// TIA Portal project "FactoryIO_Template_S7-1200_V15_V15.1" (V15.1)
// Vorlageprojekt für das Buch mit Zielsystem S7-1200

(* hardware
DEVICE "S7-1200-Station_1"  S7-1200 Station
   slot 0: "Baugruppenträger_0"  Rack  V1.0
   slot 1: "PLC_1"  CPU 1211C DC/DC/DC  6ES7 211-1AE40-0XB0  V4.1
DEVICE "HMI_1"  KTP900 Basic PN
   slot 0: "HMI_1"  KTP900 Basic PN  6AV2 123-2JB03-0AX0  15.1.0.0
   slot 1: "HMI_RT_1"  KTP900 Basic PN  6AV2 123-2JB03-0AX0  15.1.0.0
   slot 5: "HMI_1.IE_CP_1"  PROFINET Interface  15.0.1.0
      slot 1: "PROFINET Interface_1"  PROFINET Interface
         slot 1: "Port_1"  Port
*)

// ===== PLC "PLC_1"  CPU 1211C DC/DC/DC =====

VAR_GLOBAL   // PLC tag table "Standard-Variablentabelle"
   "Moving X" AT %I0.0 : Bool;
   "Moving Z" AT %I0.1 : Bool;
   "Item detected" AT %I0.2 : Bool;
   "Lid at place" AT %I0.3 : Bool;
   "Lid clamped" AT %I0.4 : Bool;
   "Pos. at limit (lids)" AT %I0.5 : Bool;
   "Base at place" AT %I0.6 : Bool;
   "Base clamped" AT %I0.7 : Bool;
   "Pos. at limit (bases)" AT %I1.0 : Bool;
   "Part leaving" AT %I1.1 : Bool;
   "Start" AT %I1.2 : Bool;
   "Reset" AT %I1.3 : Bool;
   "Stop" AT %I1.4 : Bool;
   "Emergency stop" AT %I1.5 : Bool;
   "Auto" AT %I1.6 : Bool;
   "Running" AT %I1.7 : Bool;
   "Move X" AT %Q0.0 : Bool;
   "Move Z" AT %Q0.1 : Bool;
   "Grab" AT %Q0.2 : Bool;
   "Lids conveyor" AT %Q0.3 : Bool;
   "Clamp lid" AT %Q0.4 : Bool;
   "Pos. raise (lids)" AT %Q0.5 : Bool;
   "Bases conveyor" AT %Q0.6 : Bool;
   "Clamp base" AT %Q0.7 : Bool;
   "Pos. raise (bases)" AT %Q1.0 : Bool;
   "Start light" AT %Q1.1 : Bool;
   "Reset light" AT %Q1.2 : Bool;
   "Stop light" AT %Q1.3 : Bool;
   "Counter" AT %QD30 : DInt;
END_VAR

DATA_BLOCK "Auxiliare"   // DB1
{ S7_Optimized_Access := 'TRUE' }
VERSION : 0.1
   VAR
      aux_1 : Bool;
      aux_2 : Bool;
      aux_3 : Bool;
      aux_4 : Bool;
      aux_5 : Bool;
      aux_6 : Bool;
      aux_7 : Bool;
      aux_8 : Bool;
      aux_9 : Bool;
      aux_10 : Bool;
      aux_11 : Bool;
      aux_12 : Bool;
      aux_13 : Bool;
      aux_14 : Bool;
      aux_15 : Bool;
      Lid_alined : Bool;
      Base_alined : Bool;
      Move_Z_bit : Bool;
      Move_Z_bit_2 : Bool;
      temp : Bool;
      temp_2 : Bool;
      btn_reset_counter : Bool;
   END_VAR
BEGIN
END_DATA_BLOCK

DATA_BLOCK "Alarme"   // DB3
{ S7_Optimized_Access := 'TRUE' }
VERSION : 0.1
   VAR
      esd : Bool;
   END_VAR
BEGIN
END_DATA_BLOCK

// folder: System blocks/Program resources

DATA_BLOCK "timer_grab"   // DB2
{ S7_Optimized_Access := 'TRUE' }
AUTHOR : Simatic
FAMILY : IEC
NAME : IEC_TMR
VERSION : 1.0
// stored: InstanceOfName IEC_TIMER
"IEC_TIMER"
BEGIN
END_DATA_BLOCK

DATA_BLOCK "timer_grab_2"   // DB4
{ S7_Optimized_Access := 'TRUE' }
AUTHOR : Simatic
FAMILY : IEC
NAME : IEC_TMR
VERSION : 1.0
// stored: InstanceOfName IEC_TIMER
"IEC_TIMER"
BEGIN
END_DATA_BLOCK

DATA_BLOCK "timer_ridicare_porti"   // DB5
{ S7_Optimized_Access := 'TRUE' }
AUTHOR : Simatic
FAMILY : IEC
NAME : IEC_TMR
VERSION : 1.0
// stored: InstanceOfName IEC_TIMER
"IEC_TIMER"
BEGIN
END_DATA_BLOCK

DATA_BLOCK "timer_reset_counter"   // DB6
{ S7_Optimized_Access := 'TRUE' }
AUTHOR : Simatic
FAMILY : IEC
NAME : IEC_TMR
VERSION : 1.0
// stored: InstanceOfName IEC_TIMER
"IEC_TIMER"
BEGIN
END_DATA_BLOCK

// folder: (top level)

FUNCTION "clamp" : Void   // FC1, LAD
{ S7_Optimized_Access := 'TRUE' }
VERSION : 0.1
   VAR_TEMP   // added for the SCL form of the ladder/FBD networks
      _w1 : Bool;
   END_VAR
BEGIN

REGION Network 1: clamp pentru lid
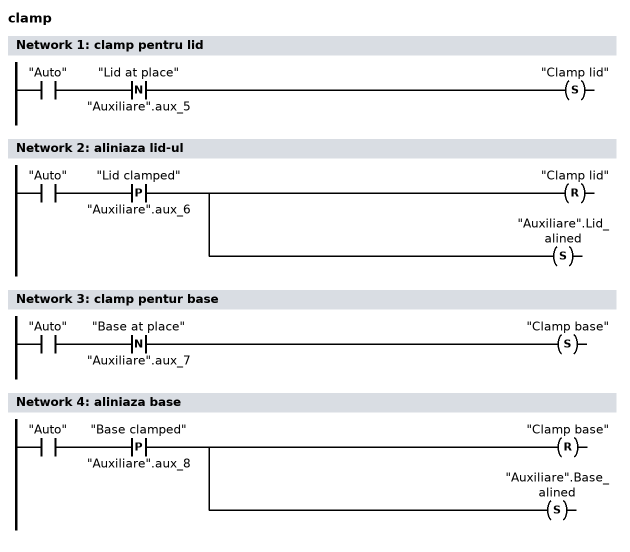
   RUNG wire#powerrail
      Contact( "Auto" )
      N_Contact(operand := "Lid at place", bit := "Auxiliare".aux_5)
      S_Coil( "Clamp lid" )
   END_RUNG
   // the same network as SCL:
   #_w1 := "Auto" AND NOT "Lid at place" AND "Auxiliare".aux_5;   // falling edge of "Lid at place"
   "Auxiliare".aux_5 := "Lid at place";
   IF #_w1 THEN "Clamp lid" := TRUE; END_IF;
END_REGION

REGION Network 2: aliniaza lid-ul
   RUNG wire#powerrail
      Contact( "Auto" )
      P_Contact(operand := "Lid clamped", bit := "Auxiliare".aux_6)
      wire#w1
      R_Coil( "Clamp lid" )
   END_RUNG
   RUNG wire#w1
      S_Coil( "Auxiliare".Lid_alined )
   END_RUNG
   // the same network as SCL:
   #_w1 := "Auto" AND "Lid clamped" AND NOT "Auxiliare".aux_6;   // rising edge of "Lid clamped"
   "Auxiliare".aux_6 := "Lid clamped";
   IF #_w1 THEN
       "Clamp lid" := FALSE;
       "Auxiliare".Lid_alined := TRUE;
   END_IF;
END_REGION

REGION Network 3: clamp pentur base
   RUNG wire#powerrail
      Contact( "Auto" )
      N_Contact(operand := "Base at place", bit := "Auxiliare".aux_7)
      S_Coil( "Clamp base" )
   END_RUNG
   // the same network as SCL:
   #_w1 := "Auto" AND NOT "Base at place" AND "Auxiliare".aux_7;   // falling edge of "Base at place"
   "Auxiliare".aux_7 := "Base at place";
   IF #_w1 THEN "Clamp base" := TRUE; END_IF;
END_REGION

REGION Network 4: aliniaza base
   RUNG wire#powerrail
      Contact( "Auto" )
      P_Contact(operand := "Base clamped", bit := "Auxiliare".aux_8)
      wire#w1
      R_Coil( "Clamp base" )
   END_RUNG
   RUNG wire#w1
      S_Coil( "Auxiliare".Base_alined )
   END_RUNG
   // the same network as SCL:
   #_w1 := "Auto" AND "Base clamped" AND NOT "Auxiliare".aux_8;   // rising edge of "Base clamped"
   "Auxiliare".aux_8 := "Base clamped";
   IF #_w1 THEN
       "Clamp base" := FALSE;
       "Auxiliare".Base_alined := TRUE;
   END_IF;
END_REGION
END_FUNCTION

FUNCTION "pick-place" : Void   // FC2, LAD
{ S7_Optimized_Access := 'TRUE' }
VERSION : 0.1
   VAR_TEMP   // added for the SCL form of the ladder/FBD networks
      _w1 : Bool;
   END_VAR
BEGIN

REGION Network 1: muta pe z ca sa ia lid ul
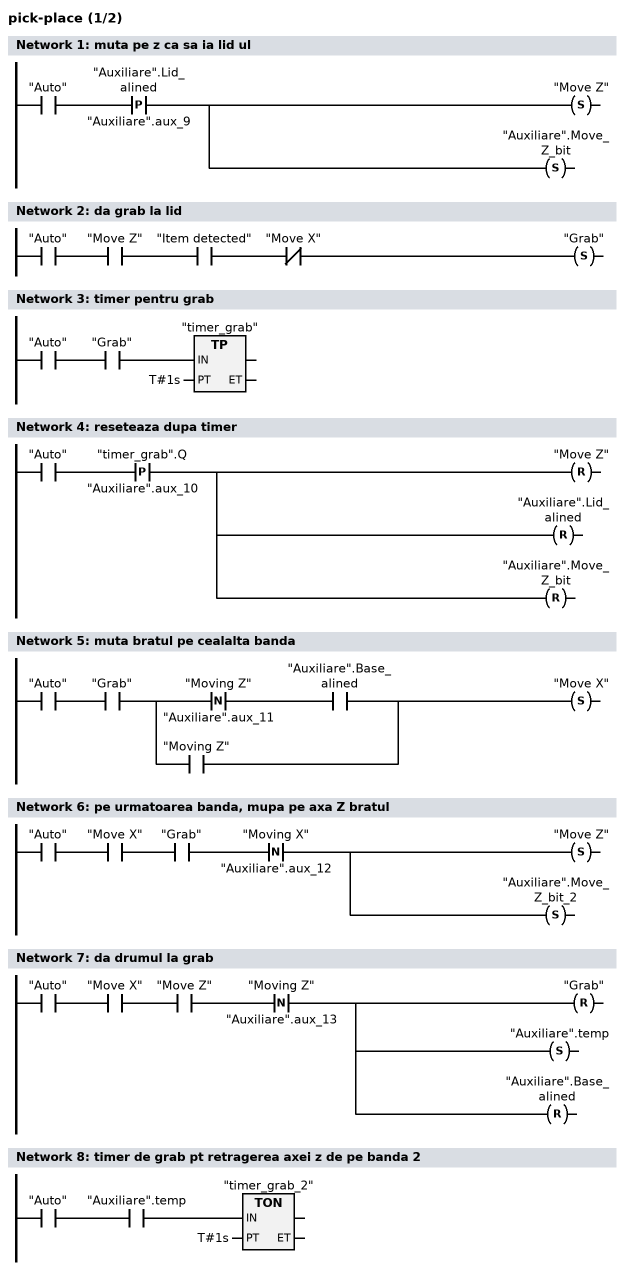
   RUNG wire#powerrail
      Contact( "Auto" )
      P_Contact(operand := "Auxiliare".Lid_alined, bit := "Auxiliare".aux_9)
      wire#w1
      S_Coil( "Move Z" )
   END_RUNG
   RUNG wire#w1
      S_Coil( "Auxiliare".Move_Z_bit )
   END_RUNG
   // the same network as SCL:
   #_w1 := "Auto" AND "Auxiliare".Lid_alined AND NOT "Auxiliare".aux_9;   // rising edge of "Auxiliare".Lid_alined
   "Auxiliare".aux_9 := "Auxiliare".Lid_alined;
   IF #_w1 THEN
       "Move Z" := TRUE;
       "Auxiliare".Move_Z_bit := TRUE;
   END_IF;
END_REGION

REGION Network 2: da grab la lid
   RUNG wire#powerrail
      Contact( "Auto" )
      Contact( "Move Z" )
      Contact( "Item detected" )
      I_Contact( "Move X" )
      S_Coil( "Grab" )
   END_RUNG
   // the same network as SCL:
   IF "Auto" AND "Move Z" AND "Item detected" AND NOT "Move X" THEN "Grab" := TRUE; END_IF;
END_REGION

REGION Network 3: timer pentru grab
   "timer_grab".TP(IN := "Auto" AND "Grab", PT := T#1s);
END_REGION

REGION Network 4: reseteaza dupa timer
   RUNG wire#powerrail
      Contact( "Auto" )
      P_Contact(operand := "timer_grab".Q, bit := "Auxiliare".aux_10)
      wire#w1
      R_Coil( "Move Z" )
   END_RUNG
   RUNG wire#w1
      R_Coil( "Auxiliare".Lid_alined )
   END_RUNG
   RUNG wire#w1
      R_Coil( "Auxiliare".Move_Z_bit )
   END_RUNG
   // the same network as SCL:
   #_w1 := "Auto" AND "timer_grab".Q AND NOT "Auxiliare".aux_10;   // rising edge of "timer_grab".Q
   "Auxiliare".aux_10 := "timer_grab".Q;
   IF #_w1 THEN
       "Move Z" := FALSE;
       "Auxiliare".Lid_alined := FALSE;
       "Auxiliare".Move_Z_bit := FALSE;
   END_IF;
END_REGION

REGION Network 5: muta bratul pe cealalta banda
   RUNG wire#powerrail
      Contact( "Auto" )
      Contact( "Grab" )
      wire#w1
      N_Contact(operand := "Moving Z", bit := "Auxiliare".aux_11)
      Contact( "Auxiliare".Base_alined )
      wire#w2
      S_Coil( "Move X" )
   END_RUNG
   RUNG wire#w1
      Contact( "Moving Z" )
   END_RUNG wire#w2
   // the same network as SCL:
   #_w1 := "Auto" AND "Grab" AND NOT "Moving Z" AND "Auxiliare".aux_11;   // falling edge of "Moving Z"
   "Auxiliare".aux_11 := "Moving Z";
   IF (#_w1 AND "Auxiliare".Base_alined) OR ("Auto" AND "Grab" AND "Moving Z") THEN "Move X" := TRUE; END_IF;
END_REGION

REGION Network 6: pe urmatoarea banda, mupa pe axa Z bratul
   RUNG wire#powerrail
      Contact( "Auto" )
      Contact( "Move X" )
      Contact( "Grab" )
      N_Contact(operand := "Moving X", bit := "Auxiliare".aux_12)
      wire#w1
      S_Coil( "Move Z" )
   END_RUNG
   RUNG wire#w1
      S_Coil( "Auxiliare".Move_Z_bit_2 )
   END_RUNG
   // the same network as SCL:
   #_w1 := "Auto" AND "Move X" AND "Grab" AND NOT "Moving X" AND "Auxiliare".aux_12;   // falling edge of "Moving X"
   "Auxiliare".aux_12 := "Moving X";
   IF #_w1 THEN
       "Move Z" := TRUE;
       "Auxiliare".Move_Z_bit_2 := TRUE;
   END_IF;
END_REGION

REGION Network 7: da drumul la grab
   RUNG wire#powerrail
      Contact( "Auto" )
      Contact( "Move X" )
      Contact( "Move Z" )
      N_Contact(operand := "Moving Z", bit := "Auxiliare".aux_13)
      wire#w1
      R_Coil( "Grab" )
   END_RUNG
   RUNG wire#w1
      S_Coil( "Auxiliare".temp )
   END_RUNG
   RUNG wire#w1
      R_Coil( "Auxiliare".Base_alined )
   END_RUNG
   // the same network as SCL:
   #_w1 := "Auto" AND "Move X" AND "Move Z" AND NOT "Moving Z" AND "Auxiliare".aux_13;   // falling edge of "Moving Z"
   "Auxiliare".aux_13 := "Moving Z";
   IF #_w1 THEN
       "Grab" := FALSE;
       "Auxiliare".temp := TRUE;
       "Auxiliare".Base_alined := FALSE;
   END_IF;
END_REGION

REGION Network 8: timer de grab pt retragerea axei z de pe banda 2
   "timer_grab_2".TON(IN := "Auto" AND "Auxiliare".temp, PT := T#1s);
END_REGION

REGION Network 9: retrage pe axa z de pe a doua banda
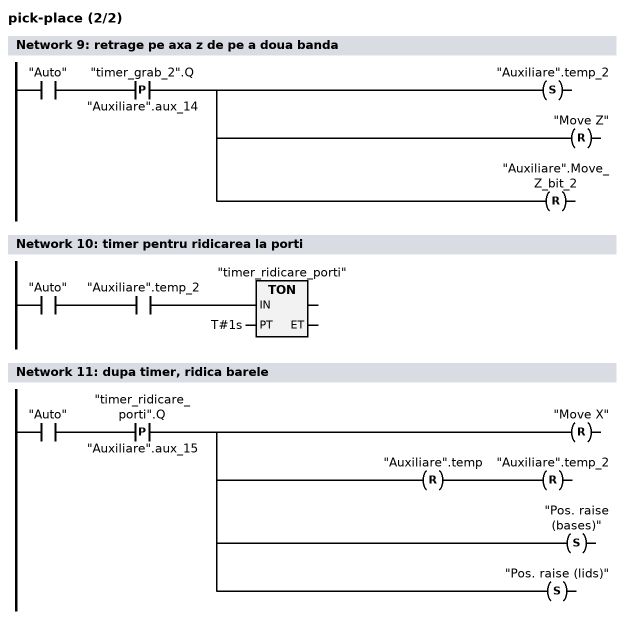
   RUNG wire#powerrail
      Contact( "Auto" )
      P_Contact(operand := "timer_grab_2".Q, bit := "Auxiliare".aux_14)
      wire#w1
      S_Coil( "Auxiliare".temp_2 )
   END_RUNG
   RUNG wire#w1
      R_Coil( "Move Z" )
   END_RUNG
   RUNG wire#w1
      R_Coil( "Auxiliare".Move_Z_bit_2 )
   END_RUNG
   // the same network as SCL:
   #_w1 := "Auto" AND "timer_grab_2".Q AND NOT "Auxiliare".aux_14;   // rising edge of "timer_grab_2".Q
   "Auxiliare".aux_14 := "timer_grab_2".Q;
   IF #_w1 THEN
       "Auxiliare".temp_2 := TRUE;
       "Move Z" := FALSE;
       "Auxiliare".Move_Z_bit_2 := FALSE;
   END_IF;
END_REGION

REGION Network 10: timer pentru ridicarea la porti
   "timer_ridicare_porti".TON(IN := "Auto" AND "Auxiliare".temp_2, PT := T#1s);
END_REGION

REGION Network 11: dupa timer, ridica barele
   RUNG wire#powerrail
      Contact( "Auto" )
      P_Contact(operand := "timer_ridicare_porti".Q, bit := "Auxiliare".aux_15)
      wire#w1
      R_Coil( "Move X" )
   END_RUNG
   RUNG wire#w1
      R_Coil( "Auxiliare".temp )
      R_Coil( "Auxiliare".temp_2 )
   END_RUNG
   RUNG wire#w1
      S_Coil( "Pos. raise (bases)" )
   END_RUNG
   RUNG wire#w1
      S_Coil( "Pos. raise (lids)" )
   END_RUNG
   // the same network as SCL:
   #_w1 := "Auto" AND "timer_ridicare_porti".Q AND NOT "Auxiliare".aux_15;   // rising edge of "timer_ridicare_porti".Q
   "Auxiliare".aux_15 := "timer_ridicare_porti".Q;
   IF #_w1 THEN
       "Move X" := FALSE;
       "Auxiliare".temp := FALSE;
       "Auxiliare".temp_2 := FALSE;
       "Pos. raise (bases)" := TRUE;
       "Pos. raise (lids)" := TRUE;
   END_IF;
END_REGION
END_FUNCTION

FUNCTION "belt" : Void   // FC3, LAD
{ S7_Optimized_Access := 'TRUE' }
VERSION : 0.1
   VAR_TEMP   // added for the SCL form of the ladder/FBD networks
      _w1 : Bool;
      _w2 : Bool;
   END_VAR
BEGIN

REGION Network 1: porneste pe auto benzile
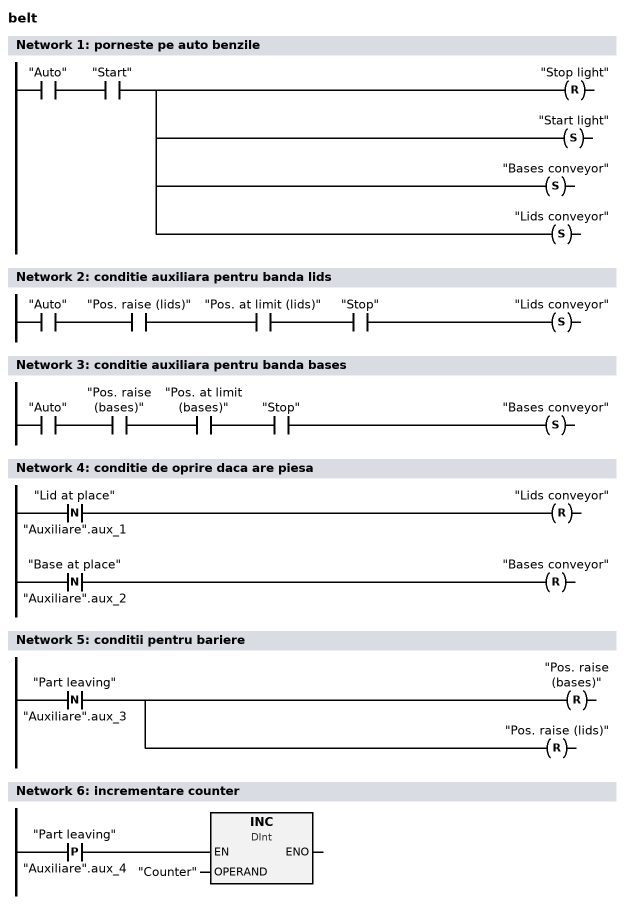
   RUNG wire#powerrail
      Contact( "Auto" )
      Contact( "Start" )
      wire#w1
      R_Coil( "Stop light" )
   END_RUNG
   RUNG wire#w1
      S_Coil( "Start light" )
   END_RUNG
   RUNG wire#w1
      S_Coil( "Bases conveyor" )
   END_RUNG
   RUNG wire#w1
      S_Coil( "Lids conveyor" )
   END_RUNG
   // the same network as SCL:
   IF "Auto" AND "Start" THEN
       "Stop light" := FALSE;
       "Start light" := TRUE;
       "Bases conveyor" := TRUE;
       "Lids conveyor" := TRUE;
   END_IF;
END_REGION

REGION Network 2: conditie auxiliara pentru banda lids
   RUNG wire#powerrail
      Contact( "Auto" )
      Contact( "Pos. raise (lids)" )
      Contact( "Pos. at limit (lids)" )
      Contact( "Stop" )
      S_Coil( "Lids conveyor" )
   END_RUNG
   // the same network as SCL:
   IF "Auto" AND "Pos. raise (lids)" AND "Pos. at limit (lids)" AND "Stop" THEN
       "Lids conveyor" := TRUE;
   END_IF;
END_REGION

REGION Network 3: conditie auxiliara pentru banda bases
   RUNG wire#powerrail
      Contact( "Auto" )
      Contact( "Pos. raise (bases)" )
      Contact( "Pos. at limit (bases)" )
      Contact( "Stop" )
      S_Coil( "Bases conveyor" )
   END_RUNG
   // the same network as SCL:
   IF "Auto" AND "Pos. raise (bases)" AND "Pos. at limit (bases)" AND "Stop" THEN
       "Bases conveyor" := TRUE;
   END_IF;
END_REGION

REGION Network 4: conditie de oprire daca are piesa
   RUNG wire#powerrail
      N_Contact(operand := "Lid at place", bit := "Auxiliare".aux_1)
      R_Coil( "Lids conveyor" )
   END_RUNG
   RUNG wire#powerrail
      N_Contact(operand := "Base at place", bit := "Auxiliare".aux_2)
      R_Coil( "Bases conveyor" )
   END_RUNG
   // the same network as SCL:
   #_w1 := NOT "Lid at place" AND "Auxiliare".aux_1;   // falling edge of "Lid at place"
   "Auxiliare".aux_1 := "Lid at place";
   IF #_w1 THEN "Lids conveyor" := FALSE; END_IF;
   #_w2 := NOT "Base at place" AND "Auxiliare".aux_2;   // falling edge of "Base at place"
   "Auxiliare".aux_2 := "Base at place";
   IF #_w2 THEN "Bases conveyor" := FALSE; END_IF;
END_REGION

REGION Network 5: conditii pentru bariere
   RUNG wire#powerrail
      N_Contact(operand := "Part leaving", bit := "Auxiliare".aux_3)
      wire#w1
      R_Coil( "Pos. raise (bases)" )
   END_RUNG
   RUNG wire#w1
      R_Coil( "Pos. raise (lids)" )
   END_RUNG
   // the same network as SCL:
   #_w1 := NOT "Part leaving" AND "Auxiliare".aux_3;   // falling edge of "Part leaving"
   "Auxiliare".aux_3 := "Part leaving";
   IF #_w1 THEN
       "Pos. raise (bases)" := FALSE;
       "Pos. raise (lids)" := FALSE;
   END_IF;
END_REGION

REGION Network 6: incrementare counter
   RUNG wire#powerrail
      P_Contact(operand := "Part leaving", bit := "Auxiliare".aux_4)
      { S7_Templates := "DestType := DInt" } Inc( "Counter" )
   END_RUNG
   // the same network as SCL:
   #_w1 := "Part leaving" AND NOT "Auxiliare".aux_4;   // rising edge of "Part leaving"
   "Auxiliare".aux_4 := "Part leaving";
   IF #_w1 THEN "Counter" := "Counter" + 1; END_IF;
END_REGION
END_FUNCTION

FUNCTION "MHJ-PLC-Lab-Function-S71200" : Void   // FC9000, SCL
{ S7_Optimized_Access := 'TRUE' }
VERSION : 0.1
   VAR_TEMP
      rdTimeReturn : Int;
      outputTime : DTL;
      SyncVal : Byte;
      forVal : Int;
      forVal_2 : Int;
      Value : Byte;
   END_VAR
   VAR CONSTANT
      CompVal : Byte := 16#34;
      Value_01 : Byte := 16#11;
      Value_01_DW : DWord := 16#A165_D992;
      Value_02_DW : DWord := 16#58BE_4401;
   END_VAR
BEGIN

   #Value:=PEEK(area := 16#82,
        dbNumber := 0,
        byteOffset := 511);
   #Value := #Value + 1;

   POKE(area := 16#82,
        dbNumber := 0,
        byteOffset := 511,
        value := #Value);

   POKE(area:=16#81,
        dbNumber:=0,
        byteOffset:=1016,
        value:=#Value_01_DW);
   POKE(area := 16#81,
        dbNumber := 0,
        byteOffset := 1020,
        value := #Value_02_DW);

   POKE(area := 16#81,
        dbNumber := 0,
        byteOffset := 511,
        value := B#16#00);

   FOR #forVal := 0 TO 120 DO
       FOR #forVal_2:=0 TO 10 DO
           #rdTimeReturn:=RD_SYS_T(#outputTime);
           #rdTimeReturn := WR_SYS_T(#outputTime);
           #rdTimeReturn := RD_SYS_T(#outputTime);
           #rdTimeReturn := WR_SYS_T(#outputTime);
       END_FOR;
       #SyncVal:= PEEK(area := 16#81,
                      dbNumber := 0,
                      byteOffset := 511);
       IF #SyncVal = #CompVal THEN
          GOTO M_1;
       END_IF;
   END_FOR;
   RETURN;

   M_1:
   POKE(area := 16#81,
        dbNumber := 0,
        byteOffset := 511,
        value := B#16#0);
END_FUNCTION

ORGANIZATION_BLOCK "Main"   // OB1, LAD, ProgramCycle
TITLE = "Main Program Sweep (Cycle)"
{ S7_Optimized_Access := 'TRUE' }
VERSION : 0.1
   VAR_INPUT
      Initial_Call : Bool;   // Initial call of this OB
      Remanence : Bool;   // =True, if remanent data are available
   END_VAR
BEGIN

REGION Network 1: Konnektierungsbaustein für PLC-Lab
   // Im Netzwerk 1 wird der Konnektierungsbaustein für PLC-Lab aufgerufen.
   // Dieser Aufruf darf nicht entfernt werden!
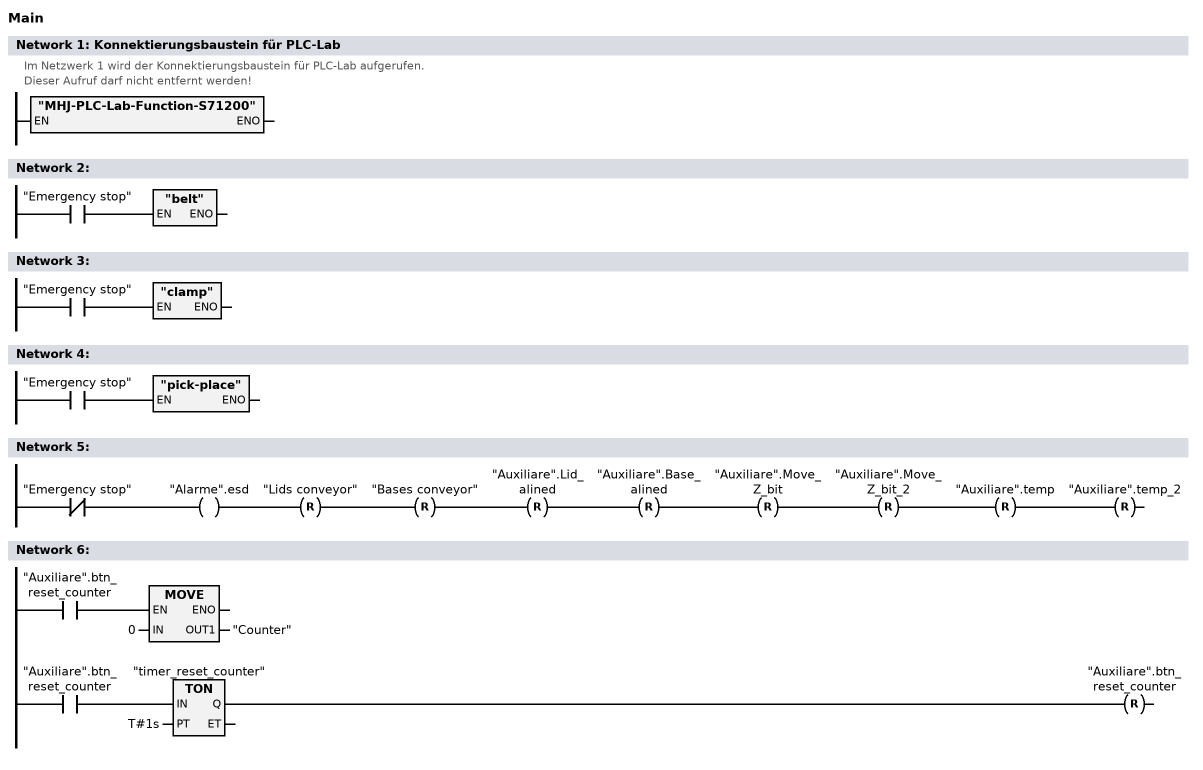
   RUNG wire#powerrail
      "MHJ-PLC-Lab-Function-S71200"()
   END_RUNG
   // the same network as SCL:
   "MHJ-PLC-Lab-Function-S71200"();
END_REGION

REGION Network 2
   RUNG wire#powerrail
      Contact( "Emergency stop" )
      "belt"()
   END_RUNG
   // the same network as SCL:
   IF "Emergency stop" THEN "belt"(); END_IF;
END_REGION

REGION Network 3
   RUNG wire#powerrail
      Contact( "Emergency stop" )
      "clamp"()
   END_RUNG
   // the same network as SCL:
   IF "Emergency stop" THEN "clamp"(); END_IF;
END_REGION

REGION Network 4
   RUNG wire#powerrail
      Contact( "Emergency stop" )
      "pick-place"()
   END_RUNG
   // the same network as SCL:
   IF "Emergency stop" THEN "pick-place"(); END_IF;
END_REGION

REGION Network 5
   RUNG wire#powerrail
      I_Contact( "Emergency stop" )
      Coil( "Alarme".esd )
      R_Coil( "Lids conveyor" )
      R_Coil( "Bases conveyor" )
      R_Coil( "Auxiliare".Lid_alined )
      R_Coil( "Auxiliare".Base_alined )
      R_Coil( "Auxiliare".Move_Z_bit )
      R_Coil( "Auxiliare".Move_Z_bit_2 )
      R_Coil( "Auxiliare".temp )
      R_Coil( "Auxiliare".temp_2 )
   END_RUNG
   // the same network as SCL:
   "Alarme".esd := NOT "Emergency stop";
   IF NOT "Emergency stop" THEN
       "Lids conveyor" := FALSE;
       "Bases conveyor" := FALSE;
       "Auxiliare".Lid_alined := FALSE;
       "Auxiliare".Base_alined := FALSE;
       "Auxiliare".Move_Z_bit := FALSE;
       "Auxiliare".Move_Z_bit_2 := FALSE;
       "Auxiliare".temp := FALSE;
       "Auxiliare".temp_2 := FALSE;
   END_IF;
END_REGION

REGION Network 6
   IF "Auxiliare".btn_reset_counter THEN "Counter" := 0; END_IF;
   "timer_reset_counter".TON(IN := "Auxiliare".btn_reset_counter, PT := T#1s);
   IF "timer_reset_counter".Q THEN "Auxiliare".btn_reset_counter := FALSE; END_IF;
END_REGION
END_ORGANIZATION_BLOCK

(* ===== HMI "HMI_RT_1" =====
system functions are stored by id; their names below are inferred from use
connection "HMI_Connection_1": ETHERNET, SMART_S7_1200_OMS

HMI tags "Default tag table"
   "running" : Bool = PLC Running AT %I1.7, 1 s
   "Alarme_esd" : Bool = PLC Alarme.esd, 1 s
   "Counter" : DInt = PLC Counter AT %QD30, 1 s
   "Auxiliare_btn_reset_counter" : Bool = PLC Auxiliare.btn_reset_counter, 1 s

Template "Template_1" 800x480
   Button "Exit" at 722,440 size 55x39; TextOff 'Exit'; PictureOff "ExitRuntime_KTP900_Basic_PN_TR"; PictureOn "ExitRuntime_KTP900_Basic_PN_TR"
      on Release: StopRuntime(0)
   Button "Template_Button" at 622,440 size 55x39; TextOff 'Text'
   Button "Template_Button_1" at 522,440 size 55x39; TextOff 'Text'
   Button "Template_Button_2" at 422,440 size 55x39; TextOff 'Text'
   Button "Template_Button_3" at 322,440 size 55x39; TextOff 'Text'
   Button "Template_Button_4" at 222,440 size 55x39; TextOff 'Text'
   Button "Template_Button_5" at 122,440 size 55x39; TextOff 'Text'
   Button "Start screen" at 22,440 size 55x39; TextOff 'Start screen'; PictureOff "NavigateHome_KTP900_Basic_PN_TR"; PictureOn "NavigateHome_KTP900_Basic_PN_TR"
      on Release: ActivateScreen("Main", 0)

screen "Main" 800x480, template "Template_1"
   IOField "I/O field_1" at 313,127 size 168x44; FormatPattern 99999
      ProcessValue <- "Counter"
   TextField "Text field_1" at 344,91 size 105x34; Text 'Counter'
   Button "Button_1" at 352,183 size 96x32; TextOff 'Reset'
      on Click: SetBit("Auxiliare_btn_reset_counter")
*)